ABB RobotStudio station: auto_calib.rspag

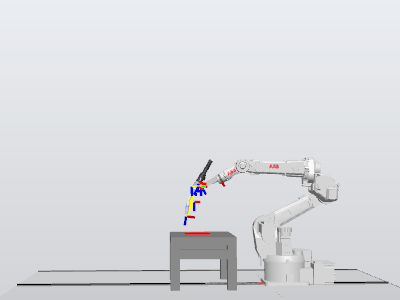
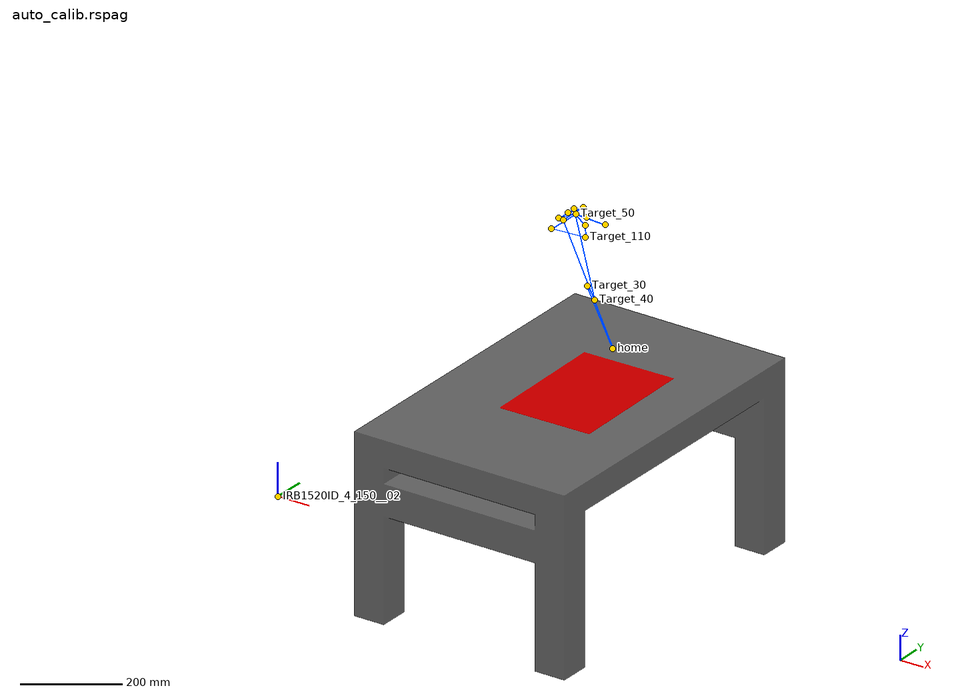
[picture v1: parts stored in the station drawn from their meshes, with robot base, taught points and paths (robot models come from the ABB library and are not in the file)]
--- station ---
Station auto_calib (saved by RobotStudio 25.5.11605.0)
Controller Controller2, task T_ROB1: task frame (RAPID world) sits at (-143.6, 0, 0) mm in the station
Controller Controller2
  mechanical unit ROB_1: IRB1520ID_4_150__02, 6 joints, base frame (0, 0, 0) mm
Layout (positions relative to the parent item):
  - IRB1520ID_4_150__02 [mechanism, from %ABB.RobotStudio.Models.IRB1520ID%\IRB1520ID_4_150_G_02.rslib] at (-143.6, 0, 0) mm; joint values [0, -1.1005, 1.0619, 0, 0.5622, 0] (rad or m)
  - Binzel_air_22 [mechanism, from %ABB.RobotStudio.Models.ArcWelding%\Binzel_air_22.rslib] at (378.41, 0, 848.1) mm, rotated rx -180 ry 60 rz -180 deg
  - Table [part] at (282.68, -348.87, 0) mm, size 500 x 750 x 400 mm
  - Paper_A4 [part] at (457.22, 184.2, 406.66) mm, rotated rx 0 ry 0 rz -88.76 deg, size 297 x 210 x 1 mm
Attachment: Binzel_air_22 is attached to IRB1520ID_4_150__02 / Link6
Attachment: Paper_A4 is attached to Table

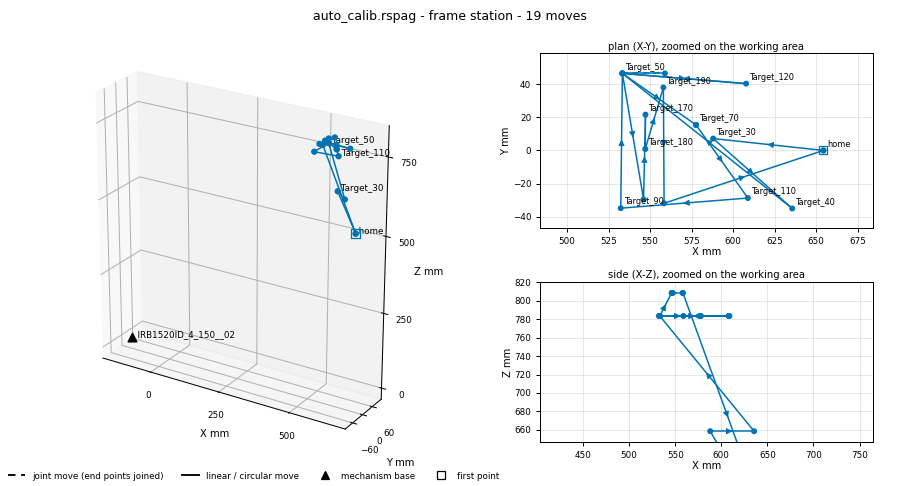
[picture p0: tool path of auto_calib.rspag in frame station, 19 of 19 moves have a stored position in this frame; points joined in program order, loops and branches not executed]
--- Backups/Controller2/RAPID/TASK1/PROGMOD/CalibData.modx ---
MODULE CalibData
    PERS tooldata tWeldGun:=[TRUE,[[125.800591275,0,391.268161315],[0.898794046,0,0.438371147,0]],[3,[0,0,100],[0,1,0,0],0,0,0]];
ENDMODULE

--- Backups/Controller2/RAPID/TASK1/PROGMOD/Module1.modx ---
MODULE Module1
    CONST robtarget home:=[[797.961954864,0,543.519411487],[0.069756473,0,0.99756405,0],[0,0,0,0],[9E+09,9E+09,9E+09,9E+09,9E+09,9E+09]];
    CONST robtarget Target_30:=[[731.572,7.169,658.548],[0,0,1,0],[0,0,0,0],[9E+09,9E+09,9E+09,9E+09,9E+09,9E+09]];
    CONST robtarget Target_40:=[[779.182,-34.96,658.548],[0,0,1,0],[0,0,0,0],[9E+09,9E+09,9E+09,9E+09,9E+09,9E+09]];
    CONST robtarget Target_50:=[[676.896972117,46.400994102,783.547920058],[-0.000000051,0.000000003,1,-0.000000008],[0,-1,0,0],[9E+09,9E+09,9E+09,9E+09,9E+09,9E+09]];
    CONST robtarget Target_70:=[[721.256,15.363,783.548],[0,0,1,0],[0,-1,0,0],[9E+09,9E+09,9E+09,9E+09,9E+09,9E+09]];
    CONST robtarget Target_110:=[[752.473,-28.67,783.548],[0,0,1,0],[-1,0,-1,0],[9E+09,9E+09,9E+09,9E+09,9E+09,9E+09]];
    CONST robtarget Target_90:=[[675.925,-34.773,783.548],[0,0,1,0],[-1,0,-1,0],[9E+09,9E+09,9E+09,9E+09,9E+09,9E+09]];
    CONST robtarget Target_100:=[[676.897,46.401,783.548],[0,0,1,0],[0,-1,0,0],[9E+09,9E+09,9E+09,9E+09,9E+09,9E+09]];
    CONST robtarget Target_120:=[[751.396,40.226,783.548],[0,0,1,0],[0,-1,0,0],[9E+09,9E+09,9E+09,9E+09,9E+09,9E+09]];
    CONST robtarget Target_160:=[[689.654,-29.507,808.548],[0,0,1,0],[-1,0,-1,0],[9E+09,9E+09,9E+09,9E+09,9E+09,9E+09]];
    CONST robtarget Target_170:=[[690.806,21.573,808.548],[0,0,1,0],[0,-1,0,0],[9E+09,9E+09,9E+09,9E+09,9E+09,9E+09]];
    CONST robtarget Target_180:=[[690.665,0.873,808.548],[0,0,1,0],[0,0,0,0],[9E+09,9E+09,9E+09,9E+09,9E+09,9E+09]];
    CONST robtarget Target_190:=[[701.596,37.931,808.548],[0,0,1,0],[0,0,0,0],[9E+09,9E+09,9E+09,9E+09,9E+09,9E+09]];
    CONST robtarget Target_200:=[[702.008,-31.805,808.548],[0,0,1,0],[0,0,0,0],[9E+09,9E+09,9E+09,9E+09,9E+09,9E+09]];
    CONST robtarget Target_50_3:=[[702.506243986,46.400994102,783.547920058],[0.220193581,0.005990523,0.974977312,0.029968998],[0,-1,0,0],[9E+09,9E+09,9E+09,9E+09,9E+09,9E+09]];
    CONST robtarget Target_50_4:=[[676.896972117,46.400994102,783.547920058],[0.267906865,-0.000000001,-0.963444815,0.000000009],[0,-1,0,0],[9E+09,9E+09,9E+09,9E+09,9E+09,9E+09]];
    CONST robtarget Target_50_2:=[[676.896972117,46.400994102,783.547920058],[-0.000000045,-0.333063821,0.942904285,-0.000000025],[-1,0,-1,0],[9E+09,9E+09,9E+09,9E+09,9E+09,9E+09]];

    PROC main()
        MoveL home,v200,fine,tWeldGun\WObj:=wobj0;
        WaitTime 3;
        MoveL Target_30,v200,fine,tWeldGun\WObj:=wobj0;
        WaitTime 3;
        MoveL Target_40,v200,fine,tWeldGun\WObj:=wobj0;
        WaitTime 3;
        MoveL Target_50,v200,fine,tWeldGun\WObj:=wobj0;
        WaitTime 3;
        MoveL Target_70,v200,fine,tWeldGun\WObj:=wobj0;
        WaitTime 3;
        MoveL Target_70,v200,fine,tWeldGun\WObj:=wobj0;
        WaitTime 3;
        MoveL Target_110,v200,fine,tWeldGun\WObj:=wobj0;
        WaitTime 3;
        MoveL Target_90,v200,fine,tWeldGun\WObj:=wobj0;
        WaitTime 3;
        MoveL Target_100,v200,fine,tWeldGun\WObj:=wobj0;
        WaitTime 3;
        MoveL Target_120,v200,fine,tWeldGun\WObj:=wobj0;
        WaitTime 3;
        MoveL Target_50_2,v200,z100,tWeldGun\WObj:=wobj0;
        WaitTime 3;
        MoveJ Target_50_3,v200,z100,tWeldGun\WObj:=wobj0;
        WaitTime 3;
        MoveL Target_50_4,v200,z100,tWeldGun\WObj:=wobj0;
        WaitTime 3;
        MoveL Target_160,v200,fine,tWeldGun\WObj:=wobj0;
        WaitTime 3;
        MoveL Target_170,v200,fine,tWeldGun\WObj:=wobj0;
        WaitTime 3;
        MoveL Target_180,v200,fine,tWeldGun\WObj:=wobj0;
        WaitTime 3;
        MoveL Target_190,v200,fine,tWeldGun\WObj:=wobj0;
        WaitTime 3;
        MoveL Target_200,v200,fine,tWeldGun\WObj:=wobj0;
        WaitTime 3;
        MoveL home,v200,fine,tWeldGun\WObj:=wobj0;
    ENDPROC
ENDMODULE

--- Backups/Controller2/SYSPAR/EIO.cfg ---
EIO:CFG_1.0:7:0::
#
VIRTUAL_NETWORK:

      -Name "Virtual" -Label "Virtual Device Network"
#
EIO_SIGNAL:

      -Name "IIO_di1" -SignalType "DI" -Device "IntegratedIOInternalDevice"\
      -DeviceMap "0"

      -Name "IIO_di2" -SignalType "DI" -Device "IntegratedIOInternalDevice"\
      -DeviceMap "1"

      -Name "IIO_di3" -SignalType "DI" -Device "IntegratedIOInternalDevice"\
      -DeviceMap "2"

      -Name "IIO_di4" -SignalType "DI" -Device "IntegratedIOInternalDevice"\
      -DeviceMap "3"

      -Name "IIO_di5" -SignalType "DI" -Device "IntegratedIOInternalDevice"\
      -DeviceMap "4"

      -Name "IIO_di6" -SignalType "DI" -Device "IntegratedIOInternalDevice"\
      -DeviceMap "5"

      -Name "IIO_di7" -SignalType "DI" -Device "IntegratedIOInternalDevice"\
      -DeviceMap "6"

      -Name "IIO_di8" -SignalType "DI" -Device "IntegratedIOInternalDevice"\
      -DeviceMap "7"

      -Name "IIO_di9" -SignalType "DI" -Device "IntegratedIOInternalDevice"\
      -DeviceMap "8"

      -Name "IIO_di10" -SignalType "DI" -Device "IntegratedIOInternalDevice"\
      -DeviceMap "9"

      -Name "IIO_di11" -SignalType "DI" -Device "IntegratedIOInternalDevice"\
      -DeviceMap "10"

      -Name "IIO_di12" -SignalType "DI" -Device "IntegratedIOInternalDevice"\
      -DeviceMap "11"

      -Name "IIO_di13" -SignalType "DI" -Device "IntegratedIOInternalDevice"\
      -DeviceMap "12"

      -Name "IIO_di14" -SignalType "DI" -Device "IntegratedIOInternalDevice"\
      -DeviceMap "13"

      -Name "IIO_di15" -SignalType "DI" -Device "IntegratedIOInternalDevice"\
      -DeviceMap "14"

      -Name "IIO_di16" -SignalType "DI" -Device "IntegratedIOInternalDevice"\
      -DeviceMap "15"

      -Name "IIO_do1" -SignalType "DO" -Device "IntegratedIOInternalDevice"\
      -DeviceMap "0"

      -Name "IIO_do2" -SignalType "DO" -Device "IntegratedIOInternalDevice"\
      -DeviceMap "1"

      -Name "IIO_do3" -SignalType "DO" -Device "IntegratedIOInternalDevice"\
      -DeviceMap "2"

      -Name "IIO_do4" -SignalType "DO" -Device "IntegratedIOInternalDevice"\
      -DeviceMap "3"

      -Name "IIO_do5" -SignalType "DO" -Device "IntegratedIOInternalDevice"\
      -DeviceMap "4"

      -Name "IIO_do6" -SignalType "DO" -Device "IntegratedIOInternalDevice"\
      -DeviceMap "5"

      -Name "IIO_do7" -SignalType "DO" -Device "IntegratedIOInternalDevice"\
      -DeviceMap "6"

      -Name "IIO_do8" -SignalType "DO" -Device "IntegratedIOInternalDevice"\
      -DeviceMap "7"

      -Name "IIO_gi" -SignalType "GI" -Device "integratedIOInternalDevice"\
      -DeviceMap "0-15"

      -Name "IIO_go" -SignalType "GO" -Device "integratedIOInternalDevice"\
      -DeviceMap "0-7"

#CTRL_SIGNATURE:YCpPdBE289rB9k8gAlEAoHs74bEIaVQb0W00eONjLiMUpGK1Yi8DJ0Sqin24DaTJK8tBghRdHOCVGnMy4bwXsw==

--- Backups/Controller2/SYSPAR/PROC.cfg ---
PROC:CFG_1.0:7:0::

#CTRL_SIGNATURE:ErYKkRYlzB2iQByPCw9d+COmI/7Z55O05k7GfQ7hGJ/xE1PPs2YQSUkPyDuwm6E78BfbtPPtnnfsrWKbyuw8+w==
